(* PLC project Unnamed, Unknown Unnamed 1 *)
(* stored: creationDateTime 2026-09-29T11:37:33, modificationDateTime 2026-09-29T14:54:44 *)

PROGRAM TankFill
  VAR
    TankFillAuto_Cmd : BOOL;
    TankValveOpen : BOOL;
    Estop_Cmd : BOOL;
    TankLevelHi_Alarm : BOOL;
    TankLevelLo_Alarm : BOOL;
    TankLevel_LIT : REAL;
    TankEmpty_SP : REAL := 2.0;
    TankFull_SP : REAL := 8.0;
    TankLoAlarm_SP : REAL := 1.0;
    TankHiAlarm_SP : REAL := 9.0;
  END_VAR

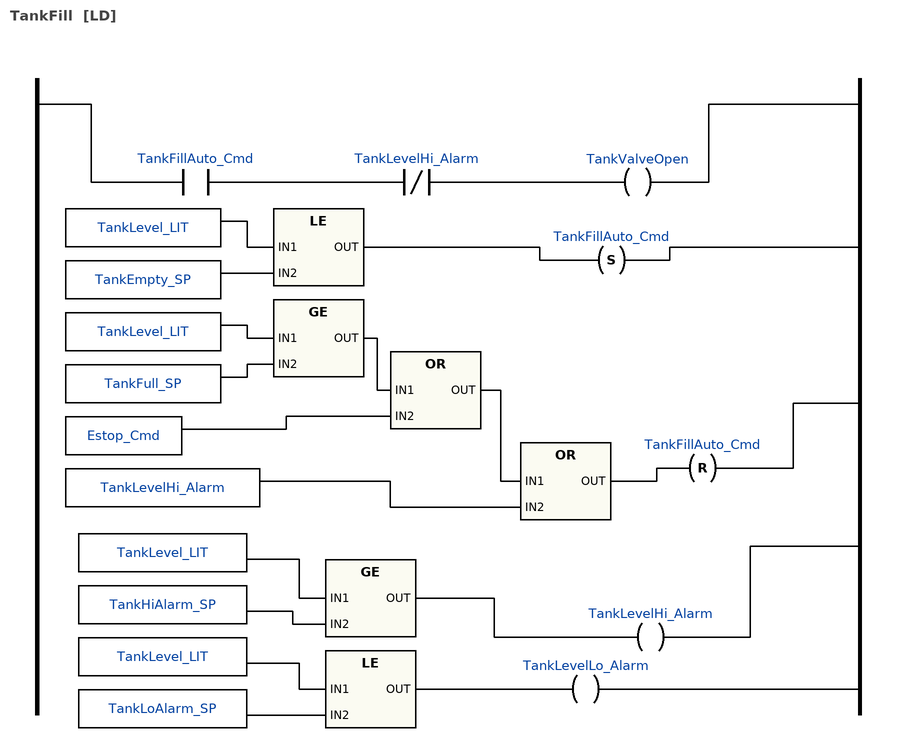
(* LD diagram, written out as Structured Text *)
TankValveOpen := TankFillAuto_Cmd AND NOT TankLevelHi_Alarm;
IF TankLevel_LIT <= TankEmpty_SP THEN TankFillAuto_Cmd := TRUE; END_IF;
TankLevelHi_Alarm := TankLevel_LIT >= TankHiAlarm_SP;
TankLevelLo_Alarm := TankLevel_LIT <= TankLoAlarm_SP;
IF TankLevel_LIT >= TankFull_SP OR Estop_Cmd OR TankLevelHi_Alarm THEN TankFillAuto_Cmd := FALSE; END_IF;
END_PROGRAM

CONFIGURATION Config0
  RESOURCE Res0 ON PLC
    TASK task0(INTERVAL := T#20ms, PRIORITY := 0);
    PROGRAM instance0 WITH task0 : TankFill;
  END_RESOURCE
END_CONFIGURATION
